PROGRAM MAIN
VAR
	bEnable : BOOL;
	bStart : BOOL;
END_VAR

bEnable := bStart;

END_PROGRAM

(* stored: Version 1.1.0.1, ProductVersion 3.1.4024.12
   POU MAIN: Id {7e5fe11e-caf9-42b9-9c2c-4a31fb34f864}, SpecialFunc None *)
